TYPE StepperSTMControl :
STRUCT
	Enable : BOOL;
	Reset : BOOL;
	ReduceTorque : BOOL;
	DigitalOutput1 : BOOL;
END_STRUCT
END_TYPE

(* stored: Version 1.1.0.1, ProductVersion 3.1.4024.9
   DUT StepperSTMControl: Id {1980a694-4cc7-4af8-9c54-18d82bbc8ff4} *)
